% RSLogix 500 project rev_pulse_1.6384b.RSS, saved by version 8.30.00.16 %
PROJECT "UNTITLED"    % processor: Bul.1763 MicroLogix 1100 Series B %

PROGRAM FILES
  LAD 2   2 rungs

DATA FILES
  O0 OUTPUT  4 elements
  I1 INPUT  6 elements
  S2 STATUS  66 elements
  B3 BINARY  24 elements
  T4 TIMER  1 elements
  C5 COUNTER  1 elements
  R6 CONTROL  1 elements
  N7 INTEGER  2 elements
  F8 FLOAT  1 elements
  L9 MISCELLANY  4 elements

LADDER 2
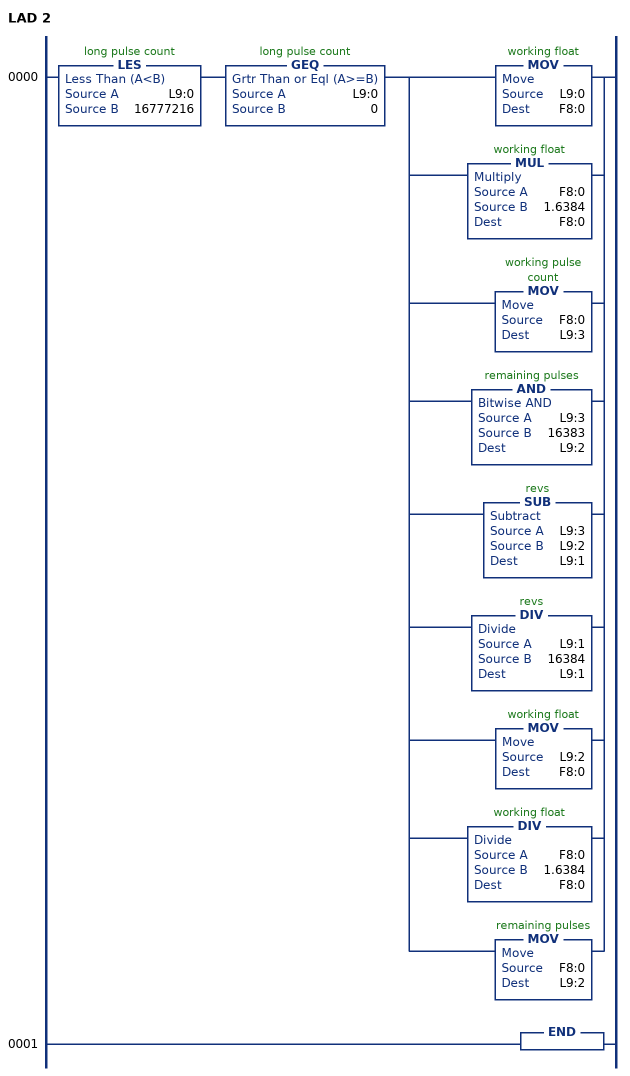
% Rung: 0 %
SOR LES L9:0 16777216 GEQ L9:0 0 BST MOV L9:0 F8:0 NXB MUL F8:0 1.6384 F8:0 NXB MOV F8:0 L9:3 NXB AND L9:3 16383 L9:2 NXB SUB L9:3 L9:2 L9:1 NXB DIV L9:1 16384 L9:1 NXB MOV L9:2 F8:0 NXB DIV F8:0 1.6384 F8:0 NXB MOV F8:0 L9:2 BND EOR
%   L9:0  "long pulse count" %
%   F8:0  "working float" %
%   L9:3  "working pulse count" %
%   L9:2  "remaining pulses" %
%   L9:1  "revs" %
% Rung: 1 %
SOR END EOR

OTHER DOCUMENTED ADDRESSES
  B3:0/0  "disable math"
  L9:4  "shifted divisor"
  L9:5  "shifted quotient"
  L9:6  "-1"
  Q2:0  "Monroe ka-chunk"
  S:22  S  "Maximum Observed Scan Time"
